// TIA Portal V16 export
// export: Created 2021-11-12T13:31:51.4017147Z, ExportSetting WithDefaults, DisplayName Totally Integrated Automation Portal, DisplayVersion V16 Update 3, DisplayName TIA Portal Version Control Interface, DisplayVersion V16 Update 2, DisplayName TIA Portal Openness, DisplayVersion V16 Update 3, DisplayName SINAMICS Startdrive Advanced, DisplayVersion V16 Update 5, DisplayName SINAMICS Startdrive G130, G150, S120, S150, SINAMICS MV, S210, DisplayVersion V16 Update 5, DisplayName SINAMICS Startdrive G110M, G120, G120C, G120D, G120P, G115D, DisplayVersion V16 Update 5, DisplayName STEP 7 Professional, DisplayVersion V16 Update 3, DisplayName STEP 7 Safety, DisplayVersion V16, DisplayName WinCC UA Professional, DisplayVersion V16 Update 3
DATA_BLOCK "HMI_CMD_000+UH01"   // DB2020
{ S7_Optimized_Access := 'TRUE' }
VERSION : 0.1
// stored: AutoNumber false, DBAccessibleFromOPCUA true, IsOnlyStoredInLoadMemory false, IsRetainMemResEnabled false, IsWriteProtectedInAS false, MemoryReserve 100
   VAR
      xxxxx___BinarySensors___xxxxx : Byte;
      xxxxx___BinaryOthers___xxxxx : Byte;
      "UC01-FV01_11" { S7_SetPoint := 'True'} : "UDT_CH_DI_Command";   // Přepěťová ochrana OK
      "UC01-FC01_14" { S7_SetPoint := 'True'} : "UDT_CH_DI_Command";   // Osvětlení a zásuvky 230V Nadproudová ochrana OK
      "UC01-FB01_14" { S7_SetPoint := 'True'} : "UDT_CH_DI_Command";   // Osvětlení a zásuvky 230V Napájecí a řídící rozvaděč OK
      "I100.3" { S7_SetPoint := 'True'} : "UDT_CH_DI_Command";   // Rezerva
      "I100.4" { S7_SetPoint := 'True'} : "UDT_CH_DI_Command";   // Rezerva
      "I100.5" { S7_SetPoint := 'True'} : "UDT_CH_DI_Command";   // Rezerva
      "I100.6" { S7_SetPoint := 'True'} : "UDT_CH_DI_Command";   // Rezerva
      "I100.7" { S7_SetPoint := 'True'} : "UDT_CH_DI_Command";   // Rezerva
      "100UC01-FC21_14" { S7_SetPoint := 'True'} : "UDT_CH_DI_Command";   // Napájení klimatizace Hlavní rozvaděč OK
      "UC01-EC01_14" { S7_SetPoint := 'True'} : "UDT_CH_DI_Command";   // Chlazení rozvaděče OK
      "UC01-FC22_14" { S7_SetPoint := 'True'} : "UDT_CH_DI_Command";   // Napájení 230V Centrální pult OK
      "UC01-FC23_14" { S7_SetPoint := 'True'} : "UDT_CH_DI_Command";   // Napájení klimatizace Centrální pult OK
      "UC01-FC24_14" { S7_SetPoint := 'True'} : "UDT_CH_DI_Command";   // Napájení klimatizace Centrální panel OK
      "400UC01-FC21_14" { S7_SetPoint := 'True'} : "UDT_CH_DI_Command";   // Napájení Osvětlení kamer OK
      "400UC01-FC22_14" { S7_SetPoint := 'True'} : "UDT_CH_DI_Command";   // Napájení Ventily Memtech OK
      "I101.7" { S7_SetPoint := 'True'} : "UDT_CH_DI_Command";   // Rezerva
      FC30_14 { S7_SetPoint := 'True'} : "UDT_CH_DI_Command";   // 24VDC (UPS) Jištění OK
      FC30_24 { S7_SetPoint := 'True'} : "UDT_CH_DI_Command";   // 24VDC (UPS) Zatížení < 90% OK
      "UC01-RB01_24" { S7_SetPoint := 'True'} : "UDT_CH_DI_Command";   // UPS Baterie OK
      FC50_14 { S7_SetPoint := 'True'} : "UDT_CH_DI_Command";   // 24VDC Jištění OK
      FC50_24 { S7_SetPoint := 'True'} : "UDT_CH_DI_Command";   // 24VDC Zatížení < 90% OK
      "I102.5" { S7_SetPoint := 'True'} : "UDT_CH_DI_Command";   // Rezerva
      "I102.6" { S7_SetPoint := 'True'} : "UDT_CH_DI_Command";   // Rezerva
      "I102.7" { S7_SetPoint := 'True'} : "UDT_CH_DI_Command";   // Rezerva
      xxxxx___AnalogueSensors___xxxxx : Byte;
      xxxxx___Drives___xxxxx : Byte;
      xxxxx___Other___xxxxx : Byte;
      xxxxx___Alarms___xxxxx : Byte;
      "UC01-FV01_12" { S7_SetPoint := 'True'} : "UDT_DI_Mon_Command";   // Přepěťová ochrana OK
      "UC01-FC01_15" { S7_SetPoint := 'True'} : "UDT_DI_Mon_Command";   // Osvětlení a zásuvky 230V Nadproudová ochrana OK
      "UC01-FB01_15" { S7_SetPoint := 'True'} : "UDT_DI_Mon_Command";   // Osvětlení a zásuvky 230V Napájecí a řídící rozvaděč OK
      "I100.8" { S7_SetPoint := 'True'} : "UDT_DI_Mon_Command";   // Rezerva
      "I100.9" { S7_SetPoint := 'True'} : "UDT_DI_Mon_Command";   // Rezerva
      "I100.10" { S7_SetPoint := 'True'} : "UDT_DI_Mon_Command";   // Rezerva
      "I100.11" { S7_SetPoint := 'True'} : "UDT_DI_Mon_Command";   // Rezerva
      "I100.12" { S7_SetPoint := 'True'} : "UDT_DI_Mon_Command";   // Rezerva
      "100UC01-FC21_15" { S7_SetPoint := 'True'} : "UDT_DI_Mon_Command";   // Napájení klimatizace Hlavní rozvaděč OK
      "UC01-EC01_15" { S7_SetPoint := 'True'} : "UDT_DI_Mon_Command";   // Chlazení rozvaděče OK
      "UC01-FC22_15" { S7_SetPoint := 'True'} : "UDT_DI_Mon_Command";   // Napájení 230V Centrální pult OK
      "UC01-FC23_15" { S7_SetPoint := 'True'} : "UDT_DI_Mon_Command";   // Napájení klimatizace Centrální pult OK
      "UC01-FC24_15" { S7_SetPoint := 'True'} : "UDT_DI_Mon_Command";   // Napájení klimatizace Centrální panel OK
      "400UC01-FC21_15" { S7_SetPoint := 'True'} : "UDT_DI_Mon_Command";   // Napájení Osvětlení kamer OK
      "400UC01-FC22_15" { S7_SetPoint := 'True'} : "UDT_DI_Mon_Command";   // Rezerva
      "I101.8" { S7_SetPoint := 'True'} : "UDT_DI_Mon_Command";   // Rezerva
      FC30_15 { S7_SetPoint := 'True'} : "UDT_DI_Mon_Command";   // 24VDC (UPS) Jištění OK
      FC30_25 { S7_SetPoint := 'True'} : "UDT_DI_Mon_Command";   // 24VDC (UPS) Zatížení < 90% OK
      "UC01-RB01_25" { S7_SetPoint := 'True'} : "UDT_DI_Mon_Command";   // UPS Baterie OK
      FC50_15 { S7_SetPoint := 'True'} : "UDT_DI_Mon_Command";   // 24VDC Jištění OK
      FC50_25 { S7_SetPoint := 'True'} : "UDT_DI_Mon_Command";   // 24VDC Zatížení < 90% OK
      "I102.8" { S7_SetPoint := 'True'} : "UDT_DI_Mon_Command";   // Rezerva
      "I102.9" { S7_SetPoint := 'True'} : "UDT_DI_Mon_Command";   // Rezerva
      "I102.10" { S7_SetPoint := 'True'} : "UDT_DI_Mon_Command";   // Rezerva
      ES { S7_SetPoint := 'True'} : "UDT_DI_Mon_Command";   // E-stop
      "000KF31" : "UDT_DI_Mon_Command";   // module 00 KF31
      "000KF32" : "UDT_DI_Mon_Command";   // module 00 KF32
      "000KF33" : "UDT_DI_Mon_Command";   // module 00 KF33
      "000KF41" : "UDT_DI_Mon_Command";   // module 00 KF41
   END_VAR
BEGIN
END_DATA_BLOCK
